PROGRAM MAIN
VAR
	fbProfiler : Profiler;
	stProfilerData : PROFILERSTRUCT;
	numFactorial : ULINT;
END_VAR

fbProfiler(START := TRUE, RESET := FALSE);
F_factorial(n := numFactorial);
fbProfiler(START := FALSE);
stProfilerData := fbProfiler.DATA;

END_PROGRAM

(* stored: Version 1.1.0.1, ProductVersion 3.1.4024.12
   POU MAIN: Id {a2a3244c-b79c-403e-8004-75bd9a7c7bef}, SpecialFunc None *)
